FUNCTION_BLOCK ModbusRTU EXTENDS Modbus
VAR_INPUT
	EN: BOOL;
END_VAR
VAR_OUTPUT
	ENO: BOOL;
END_VAR
VAR
	ModbusMaster: ModbusRtuMaster_KL6x22B;
	stMbErrId: ST_ModbusErrorDiagnostics;
	State: INT;
	aRegisterArray1: ARRAY [1..125] OF WORD;
	aRegisterCoil: ARRAY [1..250] OF BYTE;
	Param: REFERENCE TO ModbusIo;
	Delay: TON;
	StartFlag: BOOL;
	Counter: LINT;
END_VAR
VAR PERSISTENT
END_VAR

SUPER^();
ENO := EN;
Delay(IN := StartFlag, PT := T#250MS);
CASE State OF
	0:
		IF EN THEN	
			StartFlag := TRUE;	
			CurrentIoIndex := 0;
			IF IO[CurrentIoIndex] <> 0 AND Delay.Q THEN
				StartFlag := FALSE;
				State := 10;
			END_IF	
		END_IF
	10:
		Param REF= IO[CurrentIoIndex]^; 
		IF NOT Param.EN THEN
			State := 30;
		ELSE
			IF Param.RegisterType = ModbusRegisterType.Holdingregister THEN
				ModbusMaster.ReadRegs(
					UnitID := IO[CurrentIoIndex]^.UnitID, 
					Quantity := 1, 
					MBAddr := Param.Register, 
					cbLength := 2, 
					pMemoryAddr := ADR(aRegisterArray1), 
					Execute := TRUE, 
					Timeout := T#2S);
			ELSE			
				ModbusMaster.ReadInputRegs(
					UnitID := IO[CurrentIoIndex]^.UnitID, 
					Quantity := 1, 
					MBAddr := Param.Register, 
					cbLength := 2, 
					pMemoryAddr := ADR(aRegisterArray1), 
					Execute := TRUE, 
					Timeout := T#2S);
			END_IF
			IF  ModbusMaster.BUSY THEN
				State := 11;
			END_IF
		END_IF
	11:
		IF Param.RegisterType = ModbusRegisterType.Holdingregister THEN
			ModbusMaster.ReadRegs();
		ELSE
			ModbusMaster.ReadInputRegs();
		END_IF
		IF  ModbusMaster.Error or NOT ModbusMaster.BUSY THEN
			State := 20;
		END_IF
	20:
		IF Param.RegisterType = ModbusRegisterType.Holdingregister THEN
			ModbusMaster.ReadRegs();
		ELSE
			ModbusMaster.ReadInputRegs();
		END_IF
		IF ModbusMaster.Error THEN
			stMbErrId := ModbusMaster.ErrorDiagnostics;
			IF Param.RegisterType = ModbusRegisterType.Holdingregister THEN
				ModbusMaster.ReadRegs(Execute := FALSE);
			ELSE
				ModbusMaster.ReadInputRegs(Execute := FALSE);
			END_IF
			Param.ErrorOUT := TRUE;
			ErrorCount := ErrorCount + 1;
			State := 30;
		ELSIF NOT ModbusMaster.BUSY THEN
			IF Param.RegisterType = ModbusRegisterType.Holdingregister THEN
				ModbusMaster.ReadRegs(Execute := FALSE);
			ELSE
				ModbusMaster.ReadInputRegs(Execute := FALSE);
			END_IF
			Param.ValueWord := aRegisterArray1[1];
			Param.ErrorOUT := FALSE;
			ReadCount := ReadCount + 1;
			State := 30;
		END_IF
	30:
		Counter := Counter + 1;
		CurrentIoIndex := CurrentIoIndex + 1;
		IF CurrentIoIndex >= IO_COUNT THEN
			CurrentIoIndex := 0;
		END_IF
		IF IO[CurrentIoIndex] <> 0 THEN
			State := 10;
		ELSE				
			State := 0;
		END_IF
END_CASE

END_FUNCTION_BLOCK

(* stored: Version 1.1.0.1, ProductVersion 3.1.4024.6
   POU ModbusRTU: Id {d3df9997-51b6-4f4e-ba59-1348929a5873}, SpecialFunc None *)
